TYPE ST_VarBuffer :
STRUCT
	sValue 	  : STRING(2000);
	pAdress   : PVOID;
	diSize	  : DINT;  
	ClassType : __SYSTEM.TYPE_CLASS;
	bNumber   : BOOL;
END_STRUCT
END_TYPE

(* stored: Version 1.1.0.1, ProductVersion 3.1.4026.18
   DUT ST_VarBuffer: Id {c3f9d52e-eac7-460d-a866-e2205ed0dc36} *)
